(* Logix 5000 project; controller Message_L81 vendor 1 type 14 code 164 rev 36.11; software revision 36.00 *)

TASK MainTask (continuous, watchdog 500 ms) : MainProgram

MODULES
   Local : vendor 1 type 14 code 164 (ICP 0, rev 36.11)
      L62 : 1756-L62 (ICP 2, rev 20.19)
END_MODULES

VAR_GLOBAL   (* controller tags *)
   Instancia_MSG : MESSAGE;
        MessageParameters(ServiceCode := 16#0f68, LocalElement := Serial_data_L81[0], ...)
   Serial_data_L81 : INT[10] := ([1] := 2, [3] := 4, [5] := 6, [7] := 8, [9] := 10);
   Trigger : BOOL := 1;
END_VAR

PROGRAM MainProgram   (* main routine MainRoutine *)

ROUTINE MainRoutine   (* ladder *)
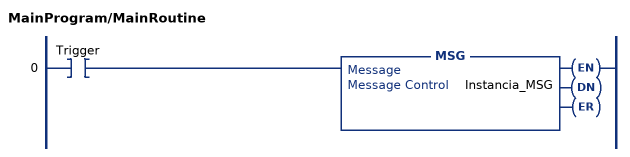
   0: XIC(Trigger)MSG(Instancia_MSG);
END_ROUTINE
END_PROGRAM
